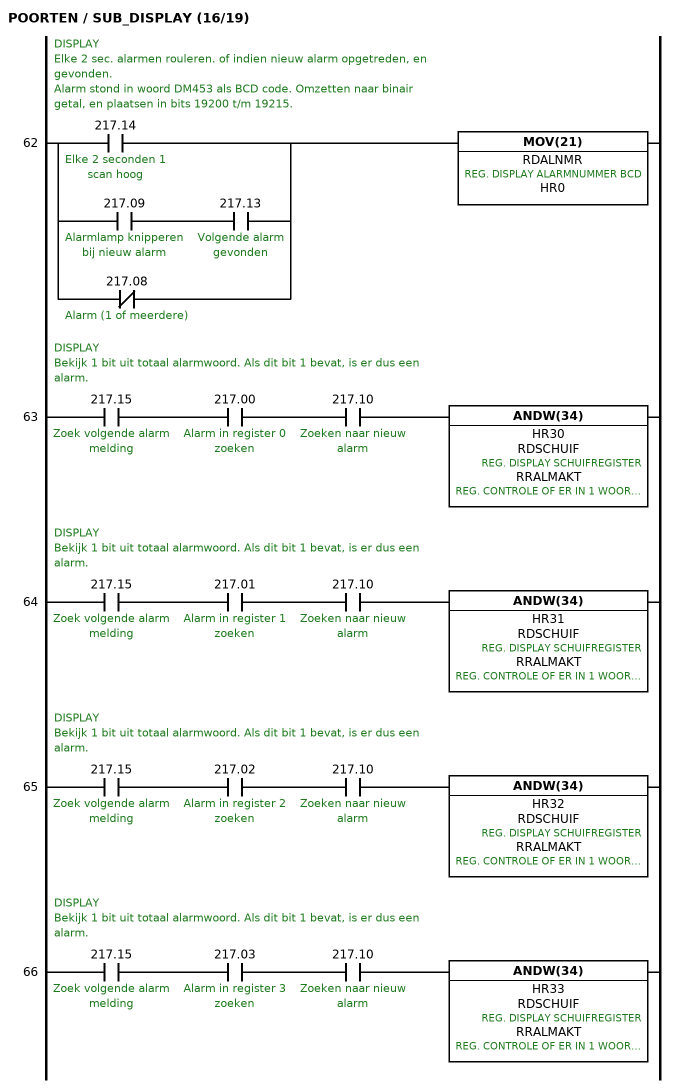
; [picture p493: POORTEN / SUB_DISPLAY, rungs 62-66]
; rung 62: DISPLAY / Elke 2 sec. alarmen rouleren. of indien nieuw alarm opgetreden, en / gevonden. / Alarm stond in woord DM453 als BCD code. Omzetten naar binair / getal, en plaatsen in bits 19200 t/m 19215.
LD 217.14  ; Elke 2 seconden 1 scan hoog
LD 217.09  ; Alarmlamp knipperen bij nieuw alarm
AND 217.13  ; Volgende alarm gevonden
ORLD
ORNOT 217.08  ; Alarm (1 of meerdere)
MOV(21) RDALNMR HR0  ; REG. DISPLAY ALARMNUMMER BCD
; rung 63: DISPLAY / Bekijk 1 bit uit totaal alarmwoord. Als dit bit 1 bevat, is er dus een / alarm.
LD 217.15  ; Zoek volgende alarm melding
AND 217.00  ; Alarm in register 0 zoeken
AND 217.10  ; Zoeken naar nieuw alarm
ANDW(34) HR30 RDSCHUIF RRALMAKT  ; REG. DISPLAY SCHUIFREGISTER, REG. CONTROLE OF ER IN 1 WOORD EEN ALARM HOOG IS
; rung 64: DISPLAY / Bekijk 1 bit uit totaal alarmwoord. Als dit bit 1 bevat, is er dus een / alarm.
LD 217.15  ; Zoek volgende alarm melding
AND 217.01  ; Alarm in register 1 zoeken
AND 217.10  ; Zoeken naar nieuw alarm
ANDW(34) HR31 RDSCHUIF RRALMAKT  ; REG. DISPLAY SCHUIFREGISTER, REG. CONTROLE OF ER IN 1 WOORD EEN ALARM HOOG IS
; rung 65: DISPLAY / Bekijk 1 bit uit totaal alarmwoord. Als dit bit 1 bevat, is er dus een / alarm.
LD 217.15  ; Zoek volgende alarm melding
AND 217.02  ; Alarm in register 2 zoeken
AND 217.10  ; Zoeken naar nieuw alarm
ANDW(34) HR32 RDSCHUIF RRALMAKT  ; REG. DISPLAY SCHUIFREGISTER, REG. CONTROLE OF ER IN 1 WOORD EEN ALARM HOOG IS
; rung 66: DISPLAY / Bekijk 1 bit uit totaal alarmwoord. Als dit bit 1 bevat, is er dus een / alarm.
LD 217.15  ; Zoek volgende alarm melding
AND 217.03  ; Alarm in register 3 zoeken
AND 217.10  ; Zoeken naar nieuw alarm
ANDW(34) HR33 RDSCHUIF RRALMAKT  ; REG. DISPLAY SCHUIFREGISTER, REG. CONTROLE OF ER IN 1 WOORD EEN ALARM HOOG IS

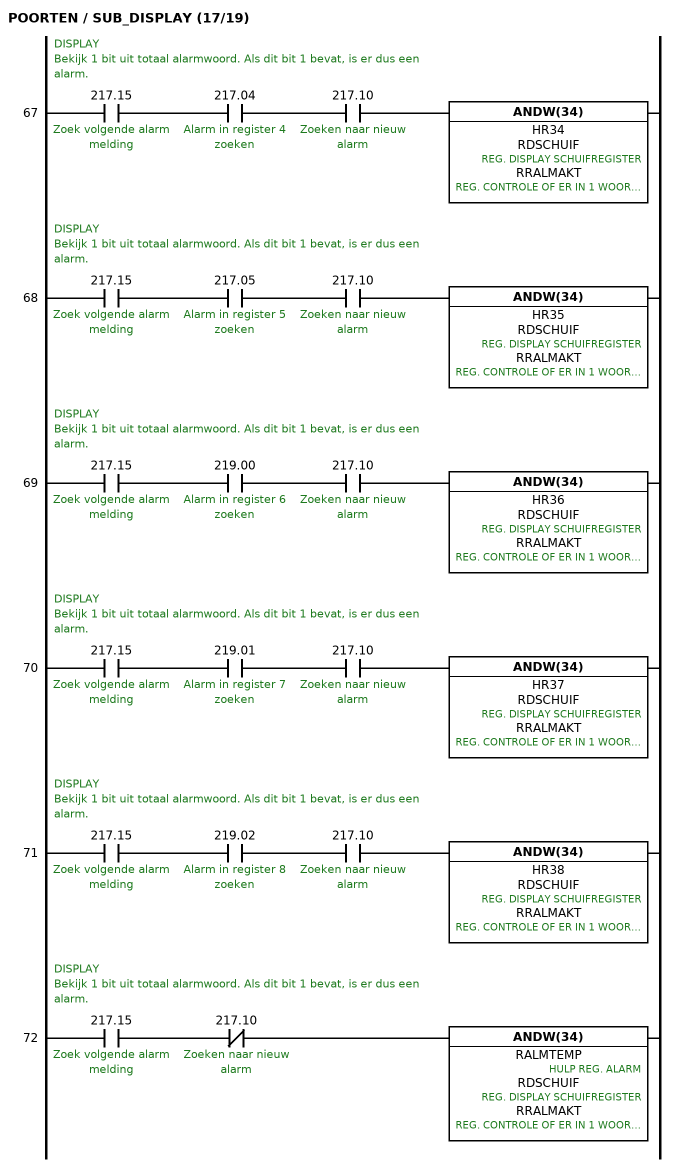
; rung 67: DISPLAY / Bekijk 1 bit uit totaal alarmwoord. Als dit bit 1 bevat, is er dus een / alarm.
LD 217.15  ; Zoek volgende alarm melding
AND 217.04  ; Alarm in register 4 zoeken
AND 217.10  ; Zoeken naar nieuw alarm
ANDW(34) HR34 RDSCHUIF RRALMAKT  ; REG. DISPLAY SCHUIFREGISTER, REG. CONTROLE OF ER IN 1 WOORD EEN ALARM HOOG IS
; rung 68: DISPLAY / Bekijk 1 bit uit totaal alarmwoord. Als dit bit 1 bevat, is er dus een / alarm.
LD 217.15  ; Zoek volgende alarm melding
AND 217.05  ; Alarm in register 5 zoeken
AND 217.10  ; Zoeken naar nieuw alarm
ANDW(34) HR35 RDSCHUIF RRALMAKT  ; REG. DISPLAY SCHUIFREGISTER, REG. CONTROLE OF ER IN 1 WOORD EEN ALARM HOOG IS
; rung 69: DISPLAY / Bekijk 1 bit uit totaal alarmwoord. Als dit bit 1 bevat, is er dus een / alarm.
LD 217.15  ; Zoek volgende alarm melding
AND 219.00  ; Alarm in register 6 zoeken
AND 217.10  ; Zoeken naar nieuw alarm
ANDW(34) HR36 RDSCHUIF RRALMAKT  ; REG. DISPLAY SCHUIFREGISTER, REG. CONTROLE OF ER IN 1 WOORD EEN ALARM HOOG IS
; rung 70: DISPLAY / Bekijk 1 bit uit totaal alarmwoord. Als dit bit 1 bevat, is er dus een / alarm.
LD 217.15  ; Zoek volgende alarm melding
AND 219.01  ; Alarm in register 7 zoeken
AND 217.10  ; Zoeken naar nieuw alarm
ANDW(34) HR37 RDSCHUIF RRALMAKT  ; REG. DISPLAY SCHUIFREGISTER, REG. CONTROLE OF ER IN 1 WOORD EEN ALARM HOOG IS
; rung 71: DISPLAY / Bekijk 1 bit uit totaal alarmwoord. Als dit bit 1 bevat, is er dus een / alarm.
LD 217.15  ; Zoek volgende alarm melding
AND 219.02  ; Alarm in register 8 zoeken
AND 217.10  ; Zoeken naar nieuw alarm
ANDW(34) HR38 RDSCHUIF RRALMAKT  ; REG. DISPLAY SCHUIFREGISTER, REG. CONTROLE OF ER IN 1 WOORD EEN ALARM HOOG IS
; rung 72: DISPLAY / Bekijk 1 bit uit totaal alarmwoord. Als dit bit 1 bevat, is er dus een / alarm.
LD 217.15  ; Zoek volgende alarm melding
ANDNOT 217.10  ; Zoeken naar nieuw alarm
ANDW(34) RALMTEMP RDSCHUIF RRALMAKT  ; HULP REG. ALARM, REG. DISPLAY SCHUIFREGISTER, REG. CONTROLE OF ER IN 1 WOORD EEN ALARM HOOG IS

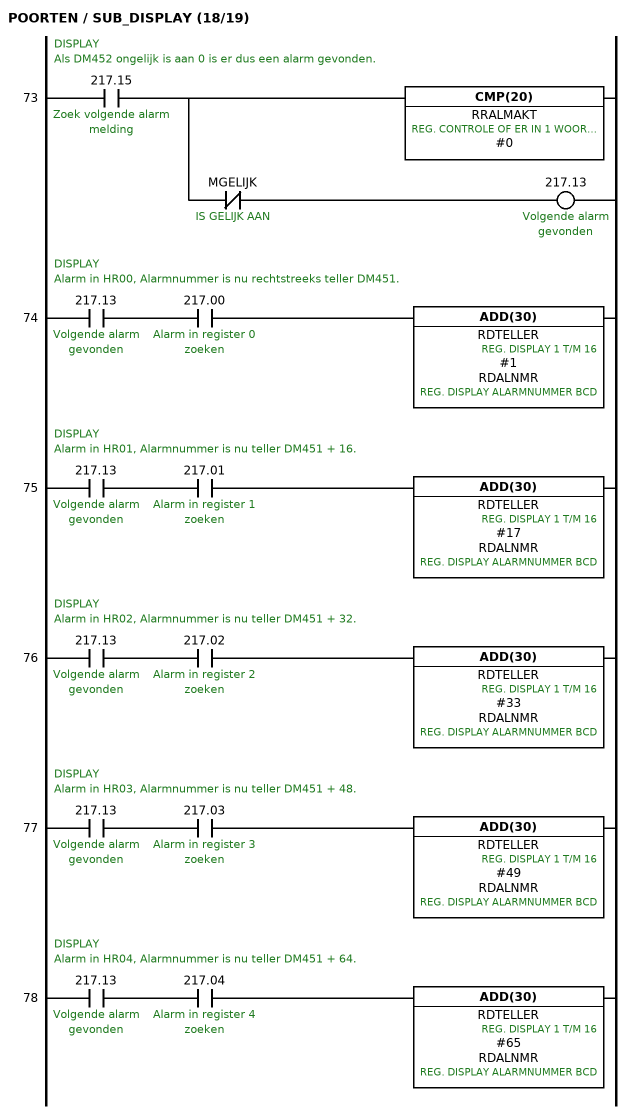
; rung 73: DISPLAY / Als DM452 ongelijk is aan 0 is er dus een alarm gevonden.
LD 217.15  ; Zoek volgende alarm melding
CMP(20) RRALMAKT #0  ; REG. CONTROLE OF ER IN 1 WOORD EEN ALARM HOOG IS
ANDNOT MGELIJK  ; IS GELIJK AAN
OUT 217.13  ; Volgende alarm gevonden
; rung 74: DISPLAY / Alarm in HR00, Alarmnummer is nu rechtstreeks teller DM451.
LD 217.13  ; Volgende alarm gevonden
AND 217.00  ; Alarm in register 0 zoeken
ADD(30) RDTELLER #1 RDALNMR  ; REG. DISPLAY 1 T/M 16, REG. DISPLAY ALARMNUMMER BCD
; rung 75: DISPLAY / Alarm in HR01, Alarmnummer is nu teller DM451 + 16.
LD 217.13  ; Volgende alarm gevonden
AND 217.01  ; Alarm in register 1 zoeken
ADD(30) RDTELLER #17 RDALNMR  ; REG. DISPLAY 1 T/M 16, REG. DISPLAY ALARMNUMMER BCD
; rung 76: DISPLAY / Alarm in HR02, Alarmnummer is nu teller DM451 + 32.
LD 217.13  ; Volgende alarm gevonden
AND 217.02  ; Alarm in register 2 zoeken
ADD(30) RDTELLER #33 RDALNMR  ; REG. DISPLAY 1 T/M 16, REG. DISPLAY ALARMNUMMER BCD
; rung 77: DISPLAY / Alarm in HR03, Alarmnummer is nu teller DM451 + 48.
LD 217.13  ; Volgende alarm gevonden
AND 217.03  ; Alarm in register 3 zoeken
ADD(30) RDTELLER #49 RDALNMR  ; REG. DISPLAY 1 T/M 16, REG. DISPLAY ALARMNUMMER BCD
; rung 78: DISPLAY / Alarm in HR04, Alarmnummer is nu teller DM451 + 64.
LD 217.13  ; Volgende alarm gevonden
AND 217.04  ; Alarm in register 4 zoeken
ADD(30) RDTELLER #65 RDALNMR  ; REG. DISPLAY 1 T/M 16, REG. DISPLAY ALARMNUMMER BCD

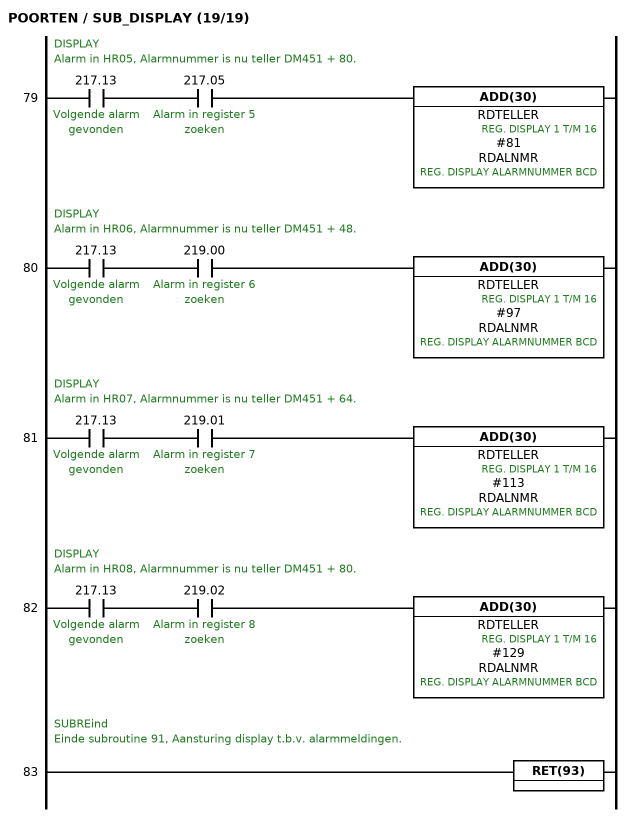
; rung 79: DISPLAY / Alarm in HR05, Alarmnummer is nu teller DM451 + 80.
LD 217.13  ; Volgende alarm gevonden
AND 217.05  ; Alarm in register 5 zoeken
ADD(30) RDTELLER #81 RDALNMR  ; REG. DISPLAY 1 T/M 16, REG. DISPLAY ALARMNUMMER BCD
; rung 80: DISPLAY / Alarm in HR06, Alarmnummer is nu teller DM451 + 48.
LD 217.13  ; Volgende alarm gevonden
AND 219.00  ; Alarm in register 6 zoeken
ADD(30) RDTELLER #97 RDALNMR  ; REG. DISPLAY 1 T/M 16, REG. DISPLAY ALARMNUMMER BCD
; rung 81: DISPLAY / Alarm in HR07, Alarmnummer is nu teller DM451 + 64.
LD 217.13  ; Volgende alarm gevonden
AND 219.01  ; Alarm in register 7 zoeken
ADD(30) RDTELLER #113 RDALNMR  ; REG. DISPLAY 1 T/M 16, REG. DISPLAY ALARMNUMMER BCD
; rung 82: DISPLAY / Alarm in HR08, Alarmnummer is nu teller DM451 + 80.
LD 217.13  ; Volgende alarm gevonden
AND 219.02  ; Alarm in register 8 zoeken
ADD(30) RDTELLER #129 RDALNMR  ; REG. DISPLAY 1 T/M 16, REG. DISPLAY ALARMNUMMER BCD
; rung 83: SUBREind / Einde subroutine 91, Aansturing display t.b.v. alarmmeldingen.
RET(93)

### Section EINDE
; rung 0: PROGR_END
END(01)